LIN {X 522.81, Y -29.184, Z 339.775, A 0, B 90, C -66.294, E1 0, E2 0, E3 0, E4 0} C_DIS
LIN {X 524.043, Y -28.836, Z 340.481, A 0, B 90, C -66.171, E1 0, E2 0, E3 0, E4 0} C_DIS
LIN {X 525.275, Y -28.481, Z 341.186, A 0, B 90, C -66.049, E1 0, E2 0, E3 0, E4 0} C_DIS
LIN {X 526.505, Y -28.118, Z 341.89, A 0, B 90, C -65.928, E1 0, E2 0, E3 0, E4 0} C_DIS
LIN {X 527.734, Y -27.747, Z 342.593, A 0, B 90, C -65.809, E1 0, E2 0, E3 0, E4 0} C_DIS
LIN {X 528.96, Y -27.369, Z 343.295, A 0, B 90, C -65.69, E1 0, E2 0, E3 0, E4 0} C_DIS
LIN {X 530.185, Y -26.983, Z 343.996, A 0, B 90, C -65.572, E1 0, E2 0, E3 0, E4 0} C_DIS
LIN {X 531.408, Y -26.589, Z 344.695, A 0, B 90, C -65.455, E1 0, E2 0, E3 0, E4 0} C_DIS
LIN {X 532.629, Y -26.187, Z 345.394, A 0, B 90, C -65.34, E1 0, E2 0, E3 0, E4 0} C_DIS
LIN {X 533.849, Y -25.778, Z 346.092, A 0, B 90, C -65.225, E1 0, E2 0, E3 0, E4 0} C_DIS
LIN {X 535.066, Y -25.361, Z 346.788, A 0, B 90, C -65.111, E1 0, E2 0, E3 0, E4 0} C_DIS
LIN {X 536.281, Y -24.936, Z 347.483, A 0, B 90, C -64.999, E1 0, E2 0, E3 0, E4 0} C_DIS
LIN {X 537.494, Y -24.504, Z 348.178, A 0, B 90, C -64.887, E1 0, E2 0, E3 0, E4 0} C_DIS
LIN {X 538.705, Y -24.064, Z 348.871, A 0, B 90, C -64.777, E1 0, E2 0, E3 0, E4 0} C_DIS
LIN {X 539.914, Y -23.617, Z 349.562, A 0, B 90, C -64.667, E1 0, E2 0, E3 0, E4 0} C_DIS
LIN {X 541.121, Y -23.162, Z 350.253, A 0, B 90, C -64.559, E1 0, E2 0, E3 0, E4 0} C_DIS
LIN {X 542.326, Y -22.699, Z 350.942, A 0, B 90, C -64.452, E1 0, E2 0, E3 0, E4 0} C_DIS
LIN {X 543.529, Y -22.229, Z 351.63, A 0, B 90, C -64.345, E1 0, E2 0, E3 0, E4 0} C_DIS
LIN {X 544.729, Y -21.751, Z 352.317, A 0, B 90, C -64.24, E1 0, E2 0, E3 0, E4 0} C_DIS
LIN {X 545.927, Y -21.266, Z 353.003, A 0, B 90, C -64.136, E1 0, E2 0, E3 0, E4 0} C_DIS
LIN {X 547.123, Y -20.773, Z 353.687, A 0, B 90, C -64.033, E1 0, E2 0, E3 0, E4 0} C_DIS
LIN {X 548.316, Y -20.273, Z 354.37, A 0, B 90, C -63.931, E1 0, E2 0, E3 0, E4 0} C_DIS
LIN {X 549.507, Y -19.765, Z 355.051, A 0, B 90, C -63.83, E1 0, E2 0, E3 0, E4 0} C_DIS
LIN {X 550.695, Y -19.25, Z 355.731, A 0, B 90, C -63.73, E1 0, E2 0, E3 0, E4 0} C_DIS
LIN {X 551.882, Y -18.727, Z 356.41, A 0, B 90, C -63.631, E1 0, E2 0, E3 0, E4 0} C_DIS
LIN {X 553.065, Y -18.197, Z 357.087, A 0, B 90, C -63.534, E1 0, E2 0, E3 0, E4 0} C_DIS
LIN {X 554.246, Y -17.659, Z 357.763, A 0, B 90, C -63.437, E1 0, E2 0, E3 0, E4 0} C_DIS
LIN {X 555.425, Y -17.114, Z 358.437, A 0, B 90, C -63.341, E1 0, E2 0, E3 0, E4 0} C_DIS
LIN {X 556.601, Y -16.561, Z 359.11, A 0, B 90, C -63.247, E1 0, E2 0, E3 0, E4 0} C_DIS
LIN {X 557.774, Y -16.001, Z 359.781, A 0, B 90, C -63.153, E1 0, E2 0, E3 0, E4 0} C_DIS
LIN {X 558.944, Y -15.434, Z 360.451, A 0, B 90, C -63.061, E1 0, E2 0, E3 0, E4 0} C_DIS
LIN {X 560.112, Y -14.86, Z 361.119, A 0, B 90, C -62.97, E1 0, E2 0, E3 0, E4 0} C_DIS
LIN {X 561.277, Y -14.278, Z 361.786, A 0, B 90, C -62.879, E1 0, E2 0, E3 0, E4 0} C_DIS
LIN {X 562.44, Y -13.688, Z 362.451, A 0, B 90, C -62.79, E1 0, E2 0, E3 0, E4 0} C_DIS
LIN {X 563.599, Y -13.092, Z 363.114, A 0, B 90, C -62.702, E1 0, E2 0, E3 0, E4 0} C_DIS
LIN {X 564.756, Y -12.488, Z 363.776, A 0, B 90, C -62.615, E1 0, E2 0, E3 0, E4 0} C_DIS
LIN {X 565.91, Y -11.877, Z 364.436, A 0, B 90, C -62.529, E1 0, E2 0, E3 0, E4 0} C_DIS
LIN {X 567.061, Y -11.258, Z 365.095, A 0, B 90, C -62.444, E1 0, E2 0, E3 0, E4 0} C_DIS
LIN {X 568.209, Y -10.633, Z 365.752, A 0, B 90, C -62.36, E1 0, E2 0, E3 0, E4 0} C_DIS
LIN {X 569.354, Y -10, Z 366.407, A 0, B 90, C -62.277, E1 0, E2 0, E3 0, E4 0} C_DIS
LIN {X 570.496, Y -9.36, Z 367.06, A 0, B 90, C -62.195, E1 0, E2 0, E3 0, E4 0} C_DIS
LIN {X 571.634, Y -8.713, Z 367.712, A 0, B 90, C -62.114, E1 0, E2 0, E3 0, E4 0} C_DIS
LIN {X 572.77, Y -8.059, Z 368.362, A 0, B 90, C -62.034, E1 0, E2 0, E3 0, E4 0} C_DIS
LIN {X 573.903, Y -7.397, Z 369.01, A 0, B 90, C -61.956, E1 0, E2 0, E3 0, E4 0} C_DIS
LIN {X 575.033, Y -6.729, Z 369.656, A 0, B 90, C -61.878, E1 0, E2 0, E3 0, E4 0} C_DIS
LIN {X 576.159, Y -6.053, Z 370.301, A 0, B 90, C -61.802, E1 0, E2 0, E3 0, E4 0} C_DIS
LIN {X 576.159, Y -6.053, Z 380.301, A 0, B 90, C -61.802, E1 0, E2 0, E3 0, E4 0}
PTP {A1 5, A2 -90, A3 100, A4 5, A5 -10, A6 -5, E1 0, E2 0, E3 0, E4 0} C_PTP
;ENDFOLD

END
